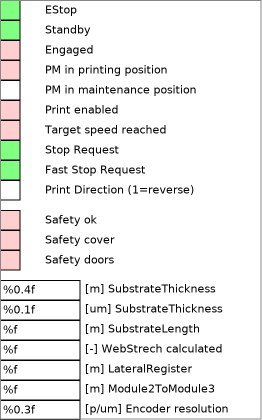
VISUALIZATION _VISU_Pm_MachineIn  // 262x420
VAR_IN_OUT
	ref : ST_ModuleMachineInterface_IN;
END_VAR
    Rectangle (0,360 80x20), "%f", text variable: ref.fLateralRegister
    Rectangle (82,360 180x18), "[m] LateralRegister"
    Rectangle (0,280 80x20), "%0.4f", text variable: ref.fSubstrateThickness
    Rectangle (82,280 180x18), "[m] SubstrateThickness"
    Rectangle (0,320 80x20), "%f", text variable: ref.fSubstrateLen
    Rectangle (82,320 180x18), "[m] SubstrateLength"
    Rectangle (0,340 80x20), "%f", text variable: ref.fWebStretchCalculated
    Rectangle (82,340 180x18), "[-] WebStrech calculated"
    Rectangle (0,380 80x20), "%f", text variable: ref.fModule2ToModule3
    Rectangle (82,380 180x18), "[m] Module2ToModule3"
    Rectangle (42,20 180x20), "Standby"
    RoundedRectangle (0,0 20x20), colour toggle: ref.bEStop
    Rectangle (42,0 180x20), "EStop"
    RoundedRectangle (0,20 20x20), colour toggle: ref.bSleep
    RoundedRectangle (0,230 20x20), colour toggle: ref.bSafetyCoverOk
    Rectangle (42,230 180x20), "Safety cover"
    RoundedRectangle (0,250 20x20), colour toggle: ref.bServiceDoorsOk
    Rectangle (42,250 180x20), "Safety doors"
    Rectangle (42,210 180x20), "Safety ok"
    RoundedRectangle (0,210 20x20), colour toggle: ref.bSafetyOk
    Rectangle (42,60 180x20), "PM in printing position"
    RoundedRectangle (0,60 20x20), colour toggle: ref.bUnitInPrintPosition
    Rectangle (42,40 180x20), "Engaged"
    RoundedRectangle (0,40 20x20), colour toggle: ref.bEngaged
    Rectangle (42,100 180x20), "Print enabled"
    RoundedRectangle (0,100 20x20), colour toggle: ref.bPrintActivated
    Rectangle (42,120 180x20), "Target speed reached"
    RoundedRectangle (0,120 20x20), colour toggle: ref.bTargetSpeedReached
    Rectangle (0,300 80x20), "%0.1f", text variable: ref.fSubstrateThickness * 1_000_000
    Rectangle (82,300 180x18), "[um] SubstrateThickness"
    Rectangle (42,140 180x20), "Stop Request"
    RoundedRectangle (0,140 20x20), colour toggle: ref.bStopRequest
    Rectangle (42,160 180x20), "Fast Stop Request"
    RoundedRectangle (0,160 20x20), colour toggle: ref.bFastStopRequest
    Rectangle (0,400 80x20), "%0.3f", text variable: ref.fEncoderResolution
    Rectangle (82,400 180x18), "[p/um] Encoder resolution"
    Rectangle (42,180 180x20), "Print Direction (1=reverse)"
    RoundedRectangle (0,180 20x20), colour toggle: ref.bPrintDirection
    Rectangle (42,80 180x20), "PM in maintenance position"
    RoundedRectangle (0,80 20x20), colour toggle: ref.bUnitInMaintPosition
END_VISUALIZATION

(* stored: Version 1.1.0.1, ProductVersion 3.1.4024.11
   Visu _VISU_Pm_MachineIn: Id {60294d81-e455-4bd4-8e0e-72ed645c373a} *)
